TYPE
    ST_MessageBox_Buttons : STRUCT
        Button1 : ST_MessageBox_Button;
        Button2 : ST_MessageBox_Button;
        Button3 : ST_MessageBox_Button;
        Button4 : ST_MessageBox_Button;
        Button5 : ST_MessageBox_Button;
    END_STRUCT
END_TYPE

(* stored: Version 1.1.0.1
   DUT ST_MessageBox_Buttons: Id {6e9466a0-6e10-44f9-a9a1-ac0e3bc0c4fb} *)
